// TIA Portal V20 export
DATA_BLOCK "DB_LoaderFixtureMain"   // DB4
// stored: InstanceOfName FB_LoaderFixtureMain, InstanceOfType FB
"FB_LoaderFixtureMain"
   // VAR
   //    sSynchroMode : Bool;
   //    sSynchroPosition : Bool;
   //    sTimeMeasure : "FB_TimeMeasure";
   //    sBlowingNotFinished { S7_SetPoint := 'True'} : Bool;
   //    sLoadingNotFinished : Bool;
   //    sUnloadingNotFinished : Bool;
   //    sReleaseNotFinished : Bool;
   //    sV_InitNotFinished : Bool;
   //    sW_InitNotFinished : Bool;
   // END_VAR
BEGIN
END_DATA_BLOCK
